Universal Robots PolyScope program: p2.urp

Program p2 (installation=default directory=/home/ur/ursim-current/programs createdIn=3.15.7.106331 lastSavedIn=3.15.7.106331 robotSerialNumber=2018339999)
Calibrated DH parameters: a=[0, -0.24365, -0.21325, 0, 0, 0]; d=[0.1519, 0, 0, 0.11235, 0.08535, 0.0819]; alpha=[1.570796, 0, 0, 1.570796, -1.570796, 0]; deltaTheta=[0, 0, 0, 0, 0, 0]
Robot Program (runOnlyOnce=true)
  Wait Sleep waitTime=9999
  MoveJ speed 60 deg/s, acceleration 80 deg/s^2 (useActiveTCP=true)
    Waypoint Waypoint_2: TCP in base x=0 y=-194.25 z=694.15 mm, rx=0 ry=2.2214 rz=-2.2214 rad; joints [0, -90, 0, -90, 0, 0] deg; pose in feature x=0 y=0 z=0 mm, rx=0 ry=0 rz=0 rad
    var_2 := MODBUS_1*(2/65535)-1
    var_3 := MODBUS_2*(2/65535)-1
    var_4 := MODBUS_3*(2/65535)-1
    var_1 := p[var_2,var_3,var_4,0,0,0]
    Waypoint Waypoint (Variable): variable=var_1
  Loop Counting (count=5) loopVariable(name=Loop_1)
    MoveL speed 250 mm/s, acceleration 1200 mm/s^2 (useActiveTCP=false) tcp=TCP; feature=Base
      MoveDirectionNode (selectedDirection=YPlus) feature=Base
        Until DISTANCE (allowActions=false deceleration=3 distanceNodeType=STOP) Distance=0.01; motionParameters(blendRadius=0)
      Wait Sleep waitTime=0.5
SubProgram SubProgram_1 (keepSynchronizedWithDisk=false)
  MoveJ speed 60 deg/s, acceleration 80 deg/s^2 (useActiveTCP=true)
    Waypoint Waypoint_2: TCP in base x=0 y=-194.25 z=694.15 mm, rx=0 ry=2.2214 rz=-2.2214 rad; joints [0, -90, 0, -90, 0, 0] deg; pose in feature x=0 y=0 z=0 mm, rx=0 ry=0 rz=0 rad
    var_2 := MODBUS_1*(10/65535)-5
    var_3 := MODBUS_2*(10/65535)-5
    var_4 := MODBUS_3*(10/65535)-5
    var_1 := p[var_2,var_3,var_4,0,0,0]
    Waypoint Waypoint (Variable): variable=var_1
    Script: write_port_register(40003,0)
Thread Thread_1 (runOnlyOnce=false)
  Wait Sleep waitTime=0.5
  Script: write_port_register(128,50)
  Wait Sleep waitTime=0.5
  Script: write_port_register(128,0)
Thread Thread_2 (runOnlyOnce=false)
  Wait Condition expression=MODBUS_5==7
  Call SubProgram_1
